FUNCTION_BLOCK FB_Error
VAR_INPUT
END_VAR
VAR_OUTPUT
END_VAR
VAR
	resetAxis			: FB_ResetAxis;
END_VAR

//@TODO: implement all possible errors

CASE errorSubState OF

	step0:	Module2301.Output.SkillOutput.SkillOutput0.Busy := FALSE;
			Module2301.Output.SkillOutput.SkillOutput0.Done := FALSE;
			Module2301.Output.SkillOutput.SkillOutput0.Dummy := FALSE;
			Module2301.Output.SkillOutput.SkillOutput0.Error := TRUE;
			Module2301.Output.SkillOutput.SkillOutput0.Ready := FALSE;
			
			//change in the right error state
			Module2301.Output.CurrentTaskDescription := 'Axis Error';
			Module2301.Output.Error := TRUE;
			
			// Error: axis got stuck
			IF (axis.Status.ErrorID = 17744) THEN
				Module2301.Output.ErrorDescription := 'Axis got stuck. Please clear module.';
				Module2301.Output.ErrorID := 301;
				errorSubState := step1;
			END_IF
			
			IF (Module2301.Output.ErrorID = 0) THEN
				Module2301.Output.ErrorDescription := 'Unknown Error.';
				Module2301.Output.ErrorID := 399;
				errorSubState := step1;
			END_IF
			
	step1:	//wait for process tool to set the module in manual mode
			IF(Module2301.Input.Mode = DUT_MODE.Manual) THEN
				resetAxis(execute:= FALSE);
				errorSubState := step2;
			END_IF
			
	step2:	IF NOT resetAxis.done THEN
				// axreset
				resetAxis (execute := TRUE);
			ELSE			
				errorSubState := step3;
			END_IF
			
	step3:	//wait for process tool to set the module in init mode
			IF(Module2301.Input.Mode = DUT_MODE.Auto) THEN
				//reset error 
				Module2301.Output.Error := FALSE;
				Module2301.Output.ErrorDescription := '';
				Module2301.Output.ErrorID := 0;
				
				//change to init state
				initSubState := step0;
				errorSubState := step0;
				mainState := eMainState.init;				
			END_IF
END_CASE

END_FUNCTION_BLOCK

(* stored: Version 1.1.0.1, ProductVersion 3.1.0.25
   POU FB_Error: Id {6c1dcf6d-4163-4cc4-8b1c-57bf0678fc07} *)
